// Mitsubishi GX Works2 project: 0624(ON_OFF스위치_PLS,FF)   PLC: Q02/Q02H

PROGRAM MAIN
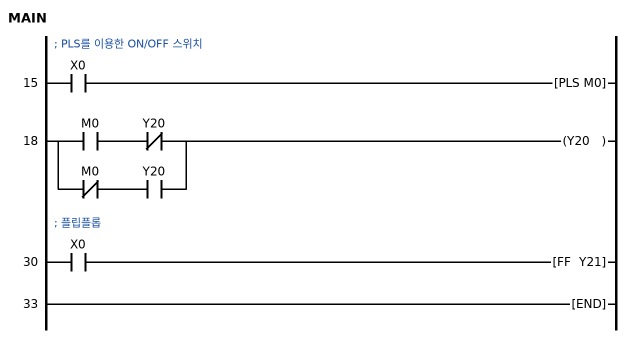
; PLS를 이용한 ON/OFF 스위치
15    LD      X0
      PLS     M0
18    LD      M0
      ANI     Y20
      LDI     M0
      AND     Y20
      ORB
      OUT     Y20
; 플립플롭
30    LD      X0
      FF      Y21
33    END
END_PROGRAM
